TYPE Coords :
STRUCT
	sName : STRING;
	iID 	: INT;
	x	: LREAL;
	y	: LREAL;
	z	: LREAL;
END_STRUCT
END_TYPE

(* stored: Version 1.1.0.1, ProductVersion 3.1.4024.11
   DUT Coords: Id {f61df51f-a098-4bd2-8db5-af9b7f2238aa} *)
